TYPE LightspeedChamberConfig EXTENDS DeviceConfiguration :
STRUCT
	{attribute 'OPC.UA.DA' := '0'}
	Version : UINT;
	{attribute 'OPC.UA.DA' := '0'}
	Description: STRING;
END_STRUCT
END_TYPE

(* stored: Version 1.1.0.1, ProductVersion 3.1.4024.12
   DUT LightspeedChamberConfig: Id {d8101e51-b516-4830-852b-9443f696806d} *)
